FUNCTION_BLOCK MOD_StateLatch (* Local channel IDs of the PackML state and its refresh query; types and forwards the received PackML state *)
  (* Standard: 61499-2 *)
  (* Version 0.1, 2026-09-28, Project contributors, AAU Smart Production Lab *)
  PACKAGE modlib;
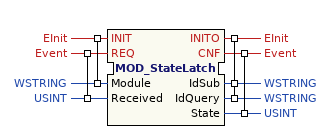
  EVENT_INPUT
    INIT : EInit WITH Module;
    REQ WITH Received;
  END_EVENT
  EVENT_OUTPUT
    INITO : EInit WITH IdSub, IdQuery;
    CNF WITH State;
  END_EVENT
  VAR_INPUT
    Module : WSTRING;
    Received : USINT;
  END_VAR
  VAR_OUTPUT
    IdSub : WSTRING;
    IdQuery : WSTRING;
    State : USINT;
  END_VAR
  EC_STATES
    INIT : INIT -> INITO;
    REQ : REQ -> CNF;
  END_STATES
  ALGORITHM INIT IN ST:
IdSub := CONCAT(CONCAT("loc[", Module), "/state]");
IdQuery := CONCAT(CONCAT("loc[", Module), "/state/query]");
  END_ALGORITHM
  ALGORITHM REQ IN ST:
State := Received;
  END_ALGORITHM
END_FUNCTION_BLOCK
